{attribute 'qualified_only'}
VAR_GLOBAL
END_VAR

(* stored: Version 1.1.0.1, ProductVersion 3.1.4024.12
   GVL G_Mode: Id {82e49624-f2a2-43d4-aee2-e5b6c8e2001e} *)
